                Wait Sleep waitTime=0.1
              IsShake := False
          Wait Sleep waitTime=0.1
    Timer (action=Stop) variable=tm_6102_01
    Set SingleDigitalPulseActionState SingleDigitalPulseActionState(hiPulseInSeconds=1, pin=GP_bool_out[15])
    Wait Sleep waitTime=1
    Popup Message (haltProgram=false message=ok? inputType=Text)
    MoveL speed 120 mm/s, acceleration 70 mm/s^2 (useActiveTCP=false) tcp=TCP_RX; feature=UF
      Waypoint Variable (Variable): variable(featureName=gGD_2_M_RX)
      Wait Sleep waitTime=1
      Waypoint Variable (Variable): variable(featureName=gGD_3_M_RX)
      Wait Sleep waitTime=1
  Folder LM
    MoveL speed 120 mm/s, acceleration 70 mm/s^2 (useActiveTCP=false) tcp=TCP_RX; feature=UF
      Waypoint Variable (Variable): variable(featureName=gGD_3_LM_RX)
      Wait Sleep waitTime=1
      Waypoint Variable (Variable): variable(featureName=gGD_2_LM_RX)
      Wait Sleep waitTime=1
      Set SingleDigitalPulseActionState SingleDigitalPulseActionState(hiPulseInSeconds=1, pin=GP_bool_out[14])
      Popup Message (haltProgram=false message=ok? inputType=Text)
    Timer (action=Reset) variable=tm_6102_01
    Timer (action=Start) variable=tm_6102_01
    SuppressedNode
      Force Frame feature=Joint_6_name; selection=[1, 1, 1, 0, 0, 0]; wrench=[0, 0, 10, 0, 0, 0]; limitsForce=[0.005, 0.005, 0.04, 0.034907, 0.034907, 1.047198]; limitsMotion=[0.1, 0.1, 0.1, 0.349066, 0.349066, 0.349066]
        Wait Condition expression=((Currpos_p_UF0[1]≤(gGD_2_LM_RX[1]-HandInZ)) or (tm_6102_01>GPII_TMHandIn))
    Timer (action=Stop) variable=tm_6102_01
    Set SingleDigitalPulseActionState SingleDigitalPulseActionState(hiPulseInSeconds=1, pin=GP_bool_out[15])
    Wait Sleep waitTime=1
    Popup Message (haltProgram=false message=ok? inputType=Text)
    MoveL speed 120 mm/s, acceleration 70 mm/s^2 (useActiveTCP=false) tcp=TCP_RX; feature=UF
      Waypoint Variable (Variable): variable(featureName=gGD_2_LM_RX)
      Wait Sleep waitTime=1
      Waypoint Variable (Variable): variable(featureName=gGD_3_LM_RX)
      Wait Sleep waitTime=1
  Folder RM
    MoveL speed 120 mm/s, acceleration 70 mm/s^2 (useActiveTCP=false) tcp=TCP_RX; feature=UF
      Waypoint Variable (Variable): variable(featureName=gGD_3_RM_RX)
      Wait Sleep waitTime=1
      Waypoint Variable (Variable): variable(featureName=gGD_2_RM_RX)
      Wait Sleep waitTime=1
      Set SingleDigitalPulseActionState SingleDigitalPulseActionState(hiPulseInSeconds=1, pin=GP_bool_out[14])
      Popup Message (haltProgram=false message=ok? inputType=Text)
    Timer (action=Reset) variable=tm_6102_01
    Timer (action=Start) variable=tm_6102_01
    SuppressedNode
      Force Frame feature=Joint_6_name; selection=[1, 1, 1, 0, 0, 0]; wrench=[0, 0, 10, 0, 0, 0]; limitsForce=[0.005, 0.005, 0.04, 0.034907, 0.034907, 1.047198]; limitsMotion=[0.1, 0.1, 0.1, 0.349066, 0.349066, 0.349066]
        Wait Condition expression=((Currpos_p_UF0[1]≤(gGD_2_RM_RX[1]-HandInZ)) or (tm_6102_01>GPII_TMHandIn))
    Timer (action=Stop) variable=tm_6102_01
    Set SingleDigitalPulseActionState SingleDigitalPulseActionState(hiPulseInSeconds=1, pin=GP_bool_out[15])
    Wait Sleep waitTime=1
    Popup Message (haltProgram=false message=ok? inputType=Text)
    MoveL speed 120 mm/s, acceleration 70 mm/s^2 (useActiveTCP=false) tcp=TCP_RX; feature=UF
      Waypoint Variable (Variable): variable(featureName=gGD_2_RM_RX)
      Wait Sleep waitTime=1
      Waypoint Variable (Variable): variable(featureName=gGD_3_RM_RX)
      Wait Sleep waitTime=1
  MoveL speed 120 mm/s, acceleration 70 mm/s^2 (useActiveTCP=false) tcp=TCP_1; feature=Base
    Waypoint Variable (Variable): variable(featureName=gHome_Position)
SubProgram SUB_6402 (keepSynchronizedWithDisk=true) programFile=/programs/GD/SUB_6402.urp
  Folder INITIALIZE
    SetPayload (workpieceName=k10)
  Folder ROVI_RECIPE
    If ( not ROVI_RECIPE(GPII_ConveyorNo))
      SubPrgResult := rovi_err
      Wait Sleep waitTime=999999
  Folder ROVI_RESET
    If ( not ROVI_RESET())
      SubPrgResult := rovi_err
      Wait Sleep waitTime=999999
  Folder ROVI_CAPTURE
    MoveL speed 200 mm/s, acceleration 70 mm/s^2 (useActiveTCP=false) tcp=TCP_1; feature=Base
      Waypoint Variable (Variable): variable(featureName=Capt_CV_M)
    Wait Sleep waitTime=2
    If ( not ROVI_CAPTURE())
      SubPrgResult := rovi_err
      Wait Sleep waitTime=999999
SubProgram SUB_7001 [hidden by the author, left out]
SubProgram SUB_7002 [hidden by the author, left out]
